// TIA Portal V17 export
// export: Created 2026-04-13T11:12:43.322584Z, ExportSetting WithDefaults, DisplayName Totally Integrated Automation Portal, DisplayVersion V17 Update 4, DisplayName TIA Portal Openness, DisplayVersion V17 Update 4, DisplayName TIA Portal Version Control Interface, DisplayVersion V17, DisplayName SINAMICS Startdrive Advanced, DisplayVersion V17, DisplayName SINAMICS Startdrive G130, G150, S120, S150, SINAMICS MV, S210, DisplayVersion V17, DisplayName SINAMICS Startdrive G110M, G120, G120C, G120D, G120P, G115D, DisplayVersion V17, DisplayName STEP 7 Professional, DisplayVersion V17 Update 4, DisplayName STEP 7 Safety, DisplayVersion V17, DisplayName WinCC Professional, DisplayVersion V17 Update 4
FUNCTION "LBitToDword" : Void   // FC231, SCL
TITLE = LBitToDWord
{ S7_Optimized_Access := 'FALSE' }
AUTHOR : Willaim
FAMILY : Control
VERSION : 0.1
// //============================================================================================
// //2017-04-21 15h49
// //Handles the conversion from bits to one DWord.
// //============================================================================================
// stored: AutoNumber false, IsIECCheckEnabled false, SetENOAutomatically false, UDAEnableTagReadback false
   VAR_INPUT
      I_Input0 : Bool;
      I_Input1 : Bool;
      I_Input2 : Bool;
      I_Input3 : Bool;
      I_Input4 : Bool;
      I_Input5 : Bool;
      I_Input6 : Bool;
      I_Input7 : Bool;
      I_Input8 : Bool;
      I_Input9 : Bool;
      I_Input10 : Bool;
      I_Input11 : Bool;
      I_Input12 : Bool;
      I_Input13 : Bool;
      I_Input14 : Bool;
      I_Input15 : Bool;
      I_Input16 : Bool;
      I_Input17 : Bool;
      I_Input18 : Bool;
      I_Input19 : Bool;
      I_Input20 : Bool;
      I_Input21 : Bool;
      I_Input22 : Bool;
      I_Input23 : Bool;
      I_Input24 : Bool;
      I_Input25 : Bool;
      I_Input26 : Bool;
      I_Input27 : Bool;
      I_Input28 : Bool;
      I_Input29 : Bool;
      I_Input30 : Bool;
      I_Input31 : Bool;
   END_VAR
   VAR_OUTPUT
      O_DWordOut : DWord;
   END_VAR
   VAR_TEMP
      TempInputBit : Array[0..31] of Bool;
      TempDWord AT TempInputBit : DWord;
   END_VAR
BEGIN
   //============================================================================================
   //2017-04-21 15h49
   //Handles the conversion from bits to one DWord.
   //============================================================================================

   //**** 1 - Inputs ****  Move Bit to temporary bit.
   #TempInputBit[24] := #I_Input0;
   #TempInputBit[25] := #I_Input1;
   #TempInputBit[26] := #I_Input2;
   #TempInputBit[27] := #I_Input3;
   #TempInputBit[28] := #I_Input4;
   #TempInputBit[29] := #I_Input5;
   #TempInputBit[30] := #I_Input6;
   #TempInputBit[31] := #I_Input7;

   #TempInputBit[16] := #I_Input8;
   #TempInputBit[17] := #I_Input9;
   #TempInputBit[18] := #I_Input10;
   #TempInputBit[19] := #I_Input11;
   #TempInputBit[20] := #I_Input12;
   #TempInputBit[21] := #I_Input13;
   #TempInputBit[22] := #I_Input14;
   #TempInputBit[23] := #I_Input15;

   #TempInputBit[8]  := #I_Input16;
   #TempInputBit[9]  := #I_Input17;
   #TempInputBit[10] := #I_Input18;
   #TempInputBit[11] := #I_Input19;
   #TempInputBit[12] := #I_Input20;
   #TempInputBit[13] := #I_Input21;
   #TempInputBit[14] := #I_Input22;
   #TempInputBit[15] := #I_Input23;

   #TempInputBit[0]  := #I_Input24;
   #TempInputBit[1]  := #I_Input25;
   #TempInputBit[2]  := #I_Input26;
   #TempInputBit[3]  := #I_Input27;
   #TempInputBit[4]  := #I_Input28;
   #TempInputBit[5]  := #I_Input29;
   #TempInputBit[6]  := #I_Input30;
   #TempInputBit[7]  := #I_Input31;

   //**** 8 - Outputs **** Move the temporary DWord to the output DWord
   #O_DWordOut := #TempDWord;
END_FUNCTION
